{attribute 'qualified_only'}
VAR_GLOBAL
	q1: REAL;
	q2  : REAL;
	q3  : REAL;
	q4 : REAL;
	q1Dot: REAL;
	q2Dot  : REAL;
	q3Dot  : REAL;
	q4Dot : REAL;
END_VAR

(* stored: Version 1.1.0.1, ProductVersion 3.1.4024.12
   GVL G_SensorsScaled: Id {fb7c7de4-6218-46cb-848a-b785536b5d86} *)
